{attribute 'GeneratedUsingTerminal: EL1918-0000-0016'}
{attribute addProperty BoxType "EL1918-0000-0016"}
{attribute addProperty Id "Module_1_FSOEModule_1_FSOE_79A9B6A834Module_2_FSLOGICModule_2_FSLOGIC_DEAB45222WcStateAT %I*WcState_9091E0EB2InfoDataAT %I*InfoData_94A18F5E2"}
{attribute addProperty CRC "3549085660"}
{attribute addProperty Size "40"}
TYPE EL1918_D38ABFDC EXTENDS EtcSlaveTerminalBase_947E5A46 :
STRUCT
	{attribute addProperty Name "Module_1_FSOE"}
	Module_1_FSOE : Module_1_FSOE_79A9B6A8;
	{attribute addProperty Name "Module_2_FSLOGIC"}
	Module_2_FSLOGIC : Module_2_FSLOGIC_DEAB4522;
	{attribute addProperty Name "WcState"}
	WcState : WcState_9091E0EB;
	{attribute addProperty Name "InfoData"}
	InfoData : InfoData_94A18F5E;
END_STRUCT
END_TYPE

(* stored: Version 1.2.0.0, ProductVersion 3.1.4024.9
   DUT EL1918_D38ABFDC: Id {eeed158b-9f9c-4c72-8cb3-d1a304af5d66} *)
